TYPE ST_Bleutooth_Status :
STRUCT
	DonglePresent 		: BIT;
	BleutoothEnabled	: BIT;
	Pairing				: BIT;
	Connected			: BIT;
	Diag				: BIT;
	InputCycleCounter	: BIT; 			
END_STRUCT
END_TYPE

(* stored: Version 1.1.0.1
   DUT ST_Bleutooth_Status: Id {a870d0e5-47d4-4843-a6c5-5c7c85d358e0} *)
